(* CoDeSys 2.3.9.59 project: ProgettoSFC.pro *)
(* Libraries: STANDARD.LIB, Iecsfc.lib 12.5.98 13:03:00 *)

(* Task configuration *)
TASK Standard (PRIORITY := 0, INTERVAL := T#10ms);
	MAIN
END_TASK

(* Global variable list: TwinCAT_Configuration *)
(* Generated automatically by TwinCAT - (read only) *)
VAR_CONFIG
	MAIN.tastatore_lettura AT %IB8 : WORD;
END_VAR

(* Data type *)
TYPE ALTEZZA: (nienteA,basso, alto);
END_TYPE

(* Data type *)
TYPE COLORE: (nienteC,rosso, altro);
END_TYPE

(* Data type *)
TYPE PEZZO :
STRUCT
	Colore : COLORE;
	Altezza : ALTEZZA;
	Trapanato:BOOL:=FALSE;
	Tastato:BOOL:=FALSE;
END_STRUCT
END_TYPE

(* Data type *)
TYPE POSTO :
STRUCT
	Presenza :BOOL:=FALSE;
	Pezzo :PEZZO;
END_STRUCT
END_TYPE

(* POU MAIN, SFC *)
PROGRAM MAIN
VAR

(*Variabili Pistone*)
         (*Ingressi*)
	pezzo_magazzino  AT%IX0.0:BOOL; (*sensore che segnala la presenza di un pezzo nel magazzino*)
	pistone_avanti AT%IX0.2:BOOL; (*sensore che segnala se il pistone è avanti*)
	pistone_indietro AT%IX0.4:BOOL; (*sensore che segnala se il pistone è indietro*)
         N_pezzi_spinti: INT:=0; (*variabile che incrementa di 1 quando viene spinto un pezzo sul nastro*)
         (*Uscite*)
	pistone_on  AT%QX0.2:BOOL; (*attuatore del pistone*)



(*Variabili Nastro*)
         (*Ingressi*)
	fine_corsa_nastro  AT%IX0.6:BOOL; (*sensore che segnala il passaggio di un pezzo a fine nastro*)
         (*Uscite*)
	nastro_on  AT%QX0.0:BOOL; (*attuatore del nastro*)


(*Variabili Giostra*)
        Giostra: ARRAY[0..7] OF POSTO;(*array di 8 posti*)
	i: INT :=0; (*indice che incrementa ad ogni movimento della giostra e usato per lavorare con l'array*)
        giostra_busy AT %IX6.1: BOOL; (*sensore che segnala il movimento della giostra*)
        movimento_giostra AT %QX3.4: BOOL; (*attuatore giostra che la muove di 1 posto*)

        T_giostra: TON; (*timer giostra di 2s*)
        mytimegiostra: TIME;
        timer_giostra: BOOL;
        reset_timer_giostra: BOOL;


        T_p1: TON; (*timer buffer 1*)
        mytimep1: TIME;
        timer_p1: BOOL;
        reset_timer_p1: BOOL;

        sensore_colore AT %IX2.1: BOOL; (*sensore che segnala i pezzi di colore rosso*)

        trapano_basso AT %IX2.5: BOOL ; (*sensore che segnala se il trapano è basso*)
        trapano_alto AT %IX2.3: BOOL; (*ensore che segnala se il trapano è alto*)
        trapano_on AT %QX3.7:BOOL; (*attuatore per l'attivazione della punta del trapano*)
        trapano_down AT %QX7.0: BOOL; (*attuatore per fare scendere o salire il trapano*)
        T_trapano: TON; (*timer trapano di 2s*)
        mytimetrapano: TIME;
        timer_trapano: BOOL;
        reset_timer_trapano: BOOL;

        tastatore_basso AT %IX5.3: BOOL; (*sensore che segnala se il tastatore è basso*)
        tastatore_alto AT %IX2.7: BOOL; (*sensore che segnala se il tastatore è alto*)
        tastatore_down AT %QX3.6: BOOL; (*attuatore tastatore*)
	tastatore_lettura AT%I*:WORD; (*fornisce la lettura dell'altezza dei pezzi*)
	(*tastatore_analogico AT %QX4.0: WORD;*)
        T_tastatore: TON; (*timer tastatore di 2s*)
        mytimetastatore: TIME;
        timer_tastatore: BOOL;
        reset_timer_tastatore: BOOL;

        pennarello_alto AT %IX5.4: BOOL; (*sensore che segnala se il pennarello è alto*)
        pennarello_basso AT %IX5.5: BOOL; (*sensore che segnala se il pennarello è basso*)
        pennarello_down AT %QX3.3: BOOL; (*attuatore pennarello*)
        T_pennarello: TON;(*timer pennarello di 2s*)
        mytimepennarello: TIME;
        timer_pennarello: BOOL;
        reset_timer_pennarello: BOOL;

        pistone_PT5_avanti AT %IX5.0: BOOL; (*sensore che segnala se il pistone 5 è avanti*)
        pistone_PT5_indietro AT %IX5.1: BOOL; (*sensore che segnala se il pistone 5 è indietro*)
        pistone_PT5_on AT %QX3.1:BOOL ; (*attuatore pistone 5*)

        pistone_PT6_avanti AT %IX5.7: BOOL;  (*sensore che segnala se il pistone 6 è avanti*)
        pistone_PT6_indietro AT %IX5.6: BOOL; (*sensore che segnala se il pistone 6 è indietro*)
        pistone_PT6_on AT%QX3.5: BOOL; (*attuatore pistone 6*)
        pezzo_baia AT %IX5.2: BOOL; (*sensore che segnala la presenza di un pezzo sulla baia*)


(*Variabili utilizzate nel FOR per la verificare alcune condizioni *)

	j: INT; (*Indice  FOR 1_posto_true*)
	posto_true: BOOL; (*Condizione di ALMENO 1 posto con presenza a TRUE*)

	k: INT; (*Indice  FOR solo_pezzi_rossi*)
	solo_pezzi_rossi: BOOL; (*Condizione SOLO pezzi rossi e  baia occupata*)

	h: INT; (*Indice FOR giostra_piena*)
	giostra_piena: BOOL; (*Condizione TUTTI i pezzi con presenza TRUE*)

	p: INT; (*Indice FOR giostra_vuota*)
	giostra_vuota: BOOL; (*Condizione se ho TUTTI i pezzi con presenza FALSE*) (*forse ridondante*)

	blocco_giostra: BOOL; (*Condizione per bloccare la giostra se ho un pezzo rosso in PT6 e la  baia è già occupata*)

	timer_pistone: BOOL;
	mytimepistone: TIME;
	reset_pistone: BOOL;
	T_pistone: TON;
	T_nastro: TON;
	mytimenastro: TIME;
	timer_nastro: BOOL;
	reset_nastro: BOOL;
	Altezza_tastatore: BOOL;
END_VAR
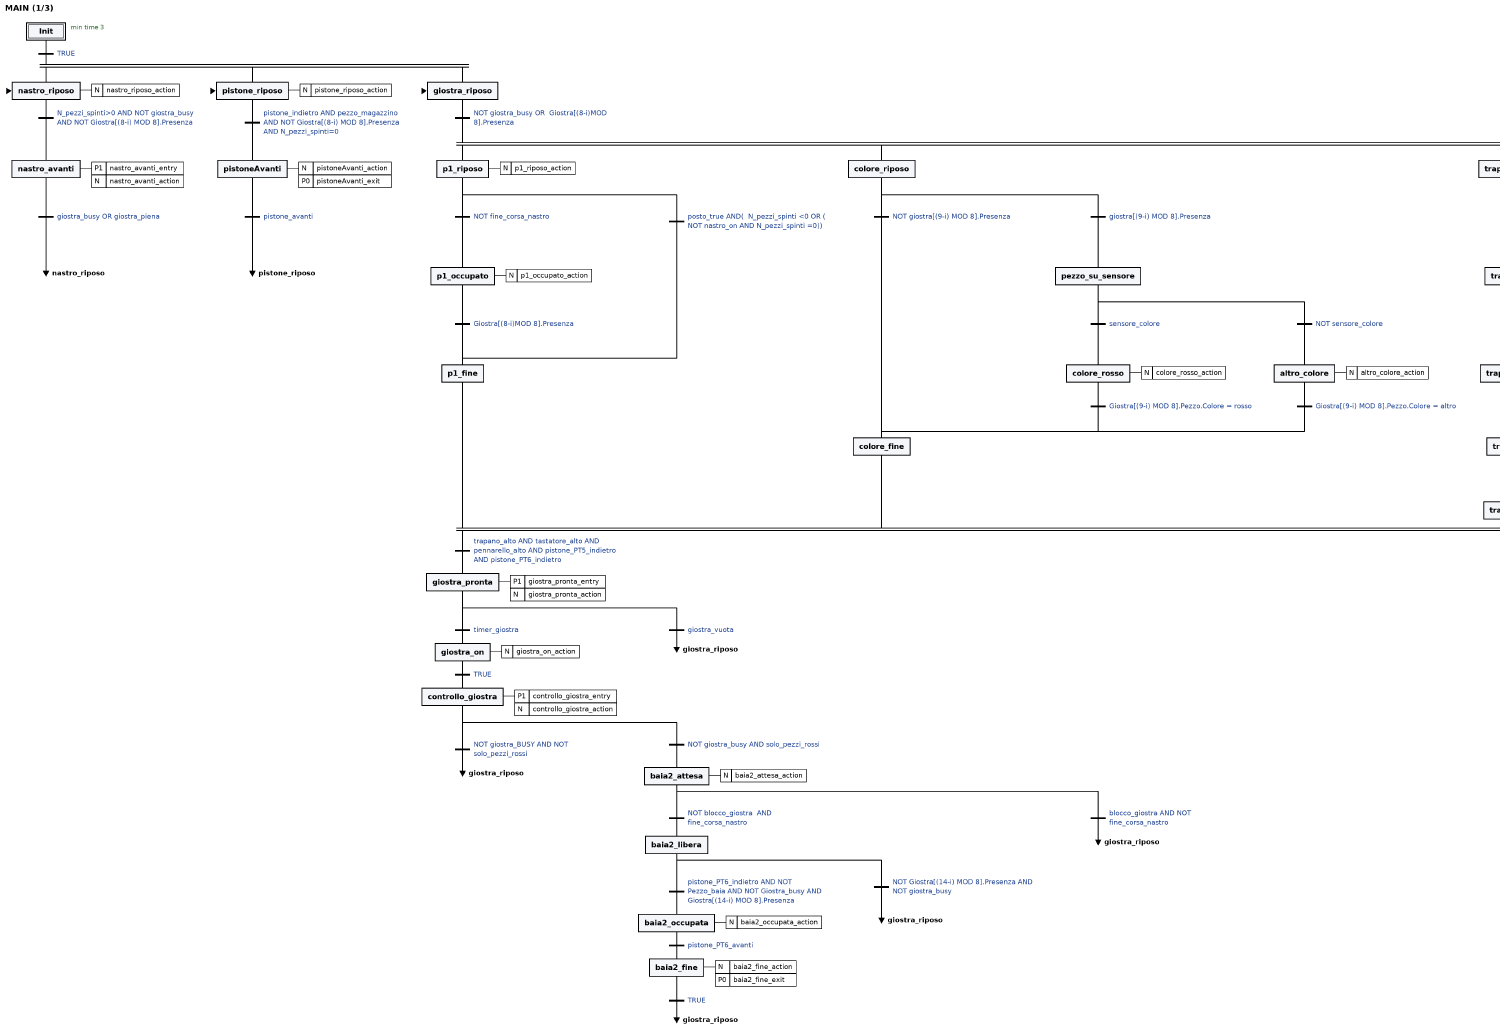
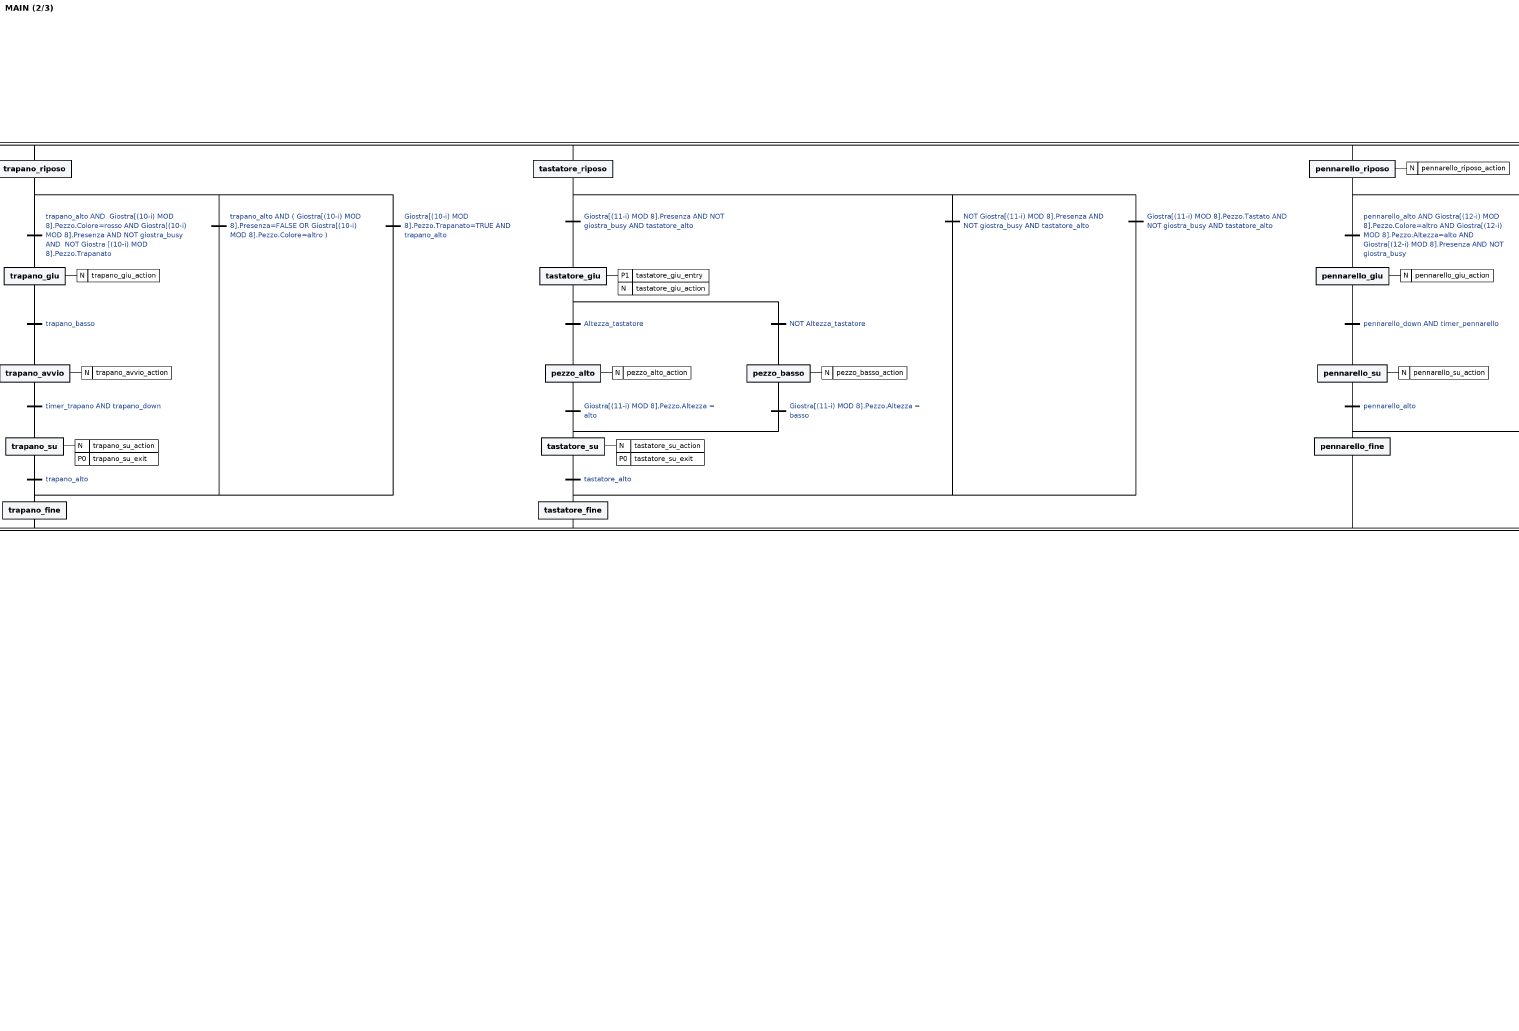
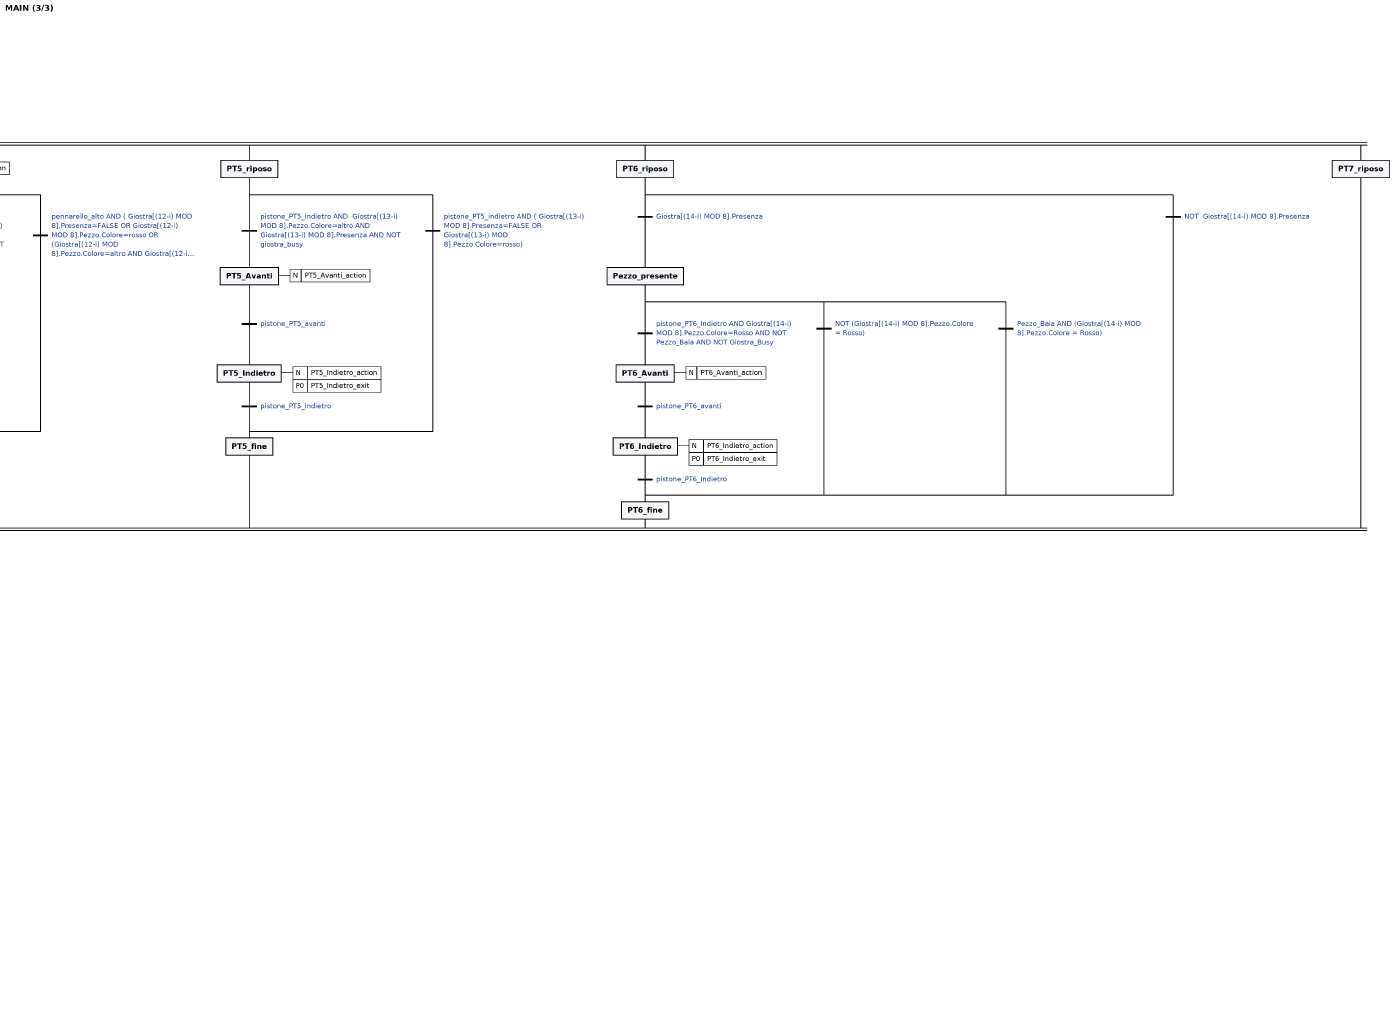
INITIAL_STEP Init: (* min time 3 *)
END_STEP
TRANSITION FROM Init TO (nastro_riposo, pistone_riposo, giostra_riposo) := TRUE;
END_TRANSITION
STEP nastro_riposo:
	nastro_riposo_action(N);
END_STEP
TRANSITION FROM nastro_riposo TO nastro_avanti := N_pezzi_spinti>0 AND NOT giostra_busy AND NOT Giostra[(8-i) MOD 8].Presenza;
END_TRANSITION
STEP pistone_riposo:
	pistone_riposo_action(N);
END_STEP
TRANSITION FROM pistone_riposo TO pistoneAvanti := pistone_indietro AND pezzo_magazzino  AND NOT Giostra[(8-i) MOD 8].Presenza AND N_pezzi_spinti=0;
END_TRANSITION
STEP giostra_riposo:
END_STEP
TRANSITION FROM giostra_riposo TO (p1_riposo, colore_riposo, trapano_riposo, tastatore_riposo, pennarello_riposo, PT5_riposo, PT6_riposo, PT7_riposo) := NOT giostra_busy OR  Giostra[(8-i)MOD 8].Presenza;
END_TRANSITION
STEP p1_riposo:
	p1_riposo_action(N);
END_STEP
TRANSITION FROM p1_riposo TO p1_occupato := NOT fine_corsa_nastro;
END_TRANSITION
TRANSITION FROM p1_riposo TO p1_fine := posto_true AND(  N_pezzi_spinti <0 OR ( NOT nastro_on AND N_pezzi_spinti =0));
END_TRANSITION
STEP p1_occupato:
	p1_occupato_action(N);
END_STEP
TRANSITION FROM p1_occupato TO p1_fine := Giostra[(8-i)MOD 8].Presenza;
END_TRANSITION
STEP p1_fine:
END_STEP
STEP colore_riposo:
END_STEP
TRANSITION FROM colore_riposo TO colore_fine := NOT giostra[(9-i) MOD 8].Presenza;
END_TRANSITION
TRANSITION FROM colore_riposo TO pezzo_su_sensore := giostra[(9-i) MOD 8].Presenza;
END_TRANSITION
STEP pezzo_su_sensore:
END_STEP
TRANSITION FROM pezzo_su_sensore TO colore_rosso := sensore_colore;
END_TRANSITION
TRANSITION FROM pezzo_su_sensore TO altro_colore := NOT sensore_colore;
END_TRANSITION
STEP colore_rosso:
	colore_rosso_action(N);
END_STEP
TRANSITION FROM colore_rosso TO colore_fine := Giostra[(9-i) MOD 8].Pezzo.Colore = rosso;
END_TRANSITION
STEP altro_colore:
	altro_colore_action(N);
END_STEP
TRANSITION FROM altro_colore TO colore_fine := Giostra[(9-i) MOD 8].Pezzo.Colore = altro;
END_TRANSITION
STEP colore_fine:
END_STEP
STEP trapano_riposo:
END_STEP
TRANSITION FROM trapano_riposo TO trapano_giu := trapano_alto AND  Giostra[(10-i) MOD 8].Pezzo.Colore=rosso AND Giostra[(10-i) MOD 8].Presenza AND NOT giostra_busy  AND  NOT Giostra [(10-i) MOD 8].Pezzo.Trapanato;
END_TRANSITION
TRANSITION FROM trapano_riposo TO trapano_fine := trapano_alto AND ( Giostra[(10-i) MOD 8].Presenza=FALSE OR Giostra[(10-i) MOD 8].Pezzo.Colore=altro );
END_TRANSITION
TRANSITION FROM trapano_riposo TO trapano_fine := Giostra[(10-i) MOD 8].Pezzo.Trapanato=TRUE AND trapano_alto;
END_TRANSITION
STEP trapano_giu:
	trapano_giu_action(N);
END_STEP
TRANSITION FROM trapano_giu TO trapano_avvio := trapano_basso;
END_TRANSITION
STEP trapano_avvio:
	trapano_avvio_action(N);
END_STEP
TRANSITION FROM trapano_avvio TO trapano_su := timer_trapano AND trapano_down;
END_TRANSITION
STEP trapano_su:
	trapano_su_action(N);
	trapano_su_exit(P0);
END_STEP
TRANSITION FROM trapano_su TO trapano_fine := trapano_alto;
END_TRANSITION
STEP trapano_fine:
END_STEP
STEP tastatore_riposo:
END_STEP
TRANSITION FROM tastatore_riposo TO tastatore_giu := Giostra[(11-i) MOD 8].Presenza AND NOT giostra_busy AND tastatore_alto;
END_TRANSITION
TRANSITION FROM tastatore_riposo TO tastatore_fine := NOT Giostra[(11-i) MOD 8].Presenza AND NOT giostra_busy AND tastatore_alto;
END_TRANSITION
TRANSITION FROM tastatore_riposo TO tastatore_fine := Giostra[(11-i) MOD 8].Pezzo.Tastato AND NOT giostra_busy AND tastatore_alto;
END_TRANSITION
STEP tastatore_giu:
	tastatore_giu_entry(P1);
	tastatore_giu_action(N);
END_STEP
TRANSITION FROM tastatore_giu TO pezzo_alto := Altezza_tastatore;
END_TRANSITION
TRANSITION FROM tastatore_giu TO pezzo_basso := NOT Altezza_tastatore;
END_TRANSITION
STEP pezzo_alto:
	pezzo_alto_action(N);
END_STEP
TRANSITION FROM pezzo_alto TO tastatore_su := Giostra[(11-i) MOD 8].Pezzo.Altezza = alto;
END_TRANSITION
STEP pezzo_basso:
	pezzo_basso_action(N);
END_STEP
TRANSITION FROM pezzo_basso TO tastatore_su := Giostra[(11-i) MOD 8].Pezzo.Altezza = basso;
END_TRANSITION
STEP tastatore_su:
	tastatore_su_action(N);
	tastatore_su_exit(P0);
END_STEP
TRANSITION FROM tastatore_su TO tastatore_fine := tastatore_alto;
END_TRANSITION
STEP tastatore_fine:
END_STEP
STEP pennarello_riposo:
	pennarello_riposo_action(N);
END_STEP
TRANSITION FROM pennarello_riposo TO pennarello_giu := pennarello_alto AND Giostra[(12-i) MOD 8].Pezzo.Colore=altro AND Giostra[(12-i) MOD 8].Pezzo.Altezza=alto AND Giostra[(12-i) MOD 8].Presenza AND NOT giostra_busy;
END_TRANSITION
TRANSITION FROM pennarello_riposo TO pennarello_fine := pennarello_alto AND ( Giostra[(12-i) MOD 8].Presenza=FALSE OR Giostra[(12-i) MOD 8].Pezzo.Colore=rosso OR (Giostra[(12-i) MOD 8].Pezzo.Colore=altro AND Giostra[(12-i) MOD 8].Pezzo.Altezza=basso));
END_TRANSITION
STEP pennarello_giu:
	pennarello_giu_action(N);
END_STEP
TRANSITION FROM pennarello_giu TO pennarello_su := pennarello_down AND timer_pennarello;
END_TRANSITION
STEP pennarello_su:
	pennarello_su_action(N);
END_STEP
TRANSITION FROM pennarello_su TO pennarello_fine := pennarello_alto;
END_TRANSITION
STEP pennarello_fine:
END_STEP
STEP PT5_riposo:
END_STEP
TRANSITION FROM PT5_riposo TO PT5_Avanti := pistone_PT5_indietro AND  Giostra[(13-i) MOD 8].Pezzo.Colore=altro AND Giostra[(13-i) MOD 8].Presenza AND NOT giostra_busy;
END_TRANSITION
TRANSITION FROM PT5_riposo TO PT5_fine := pistone_PT5_indietro AND ( Giostra[(13-i) MOD 8].Presenza=FALSE OR Giostra[(13-i) MOD 8].Pezzo.Colore=rosso);
END_TRANSITION
STEP PT5_Avanti:
	PT5_Avanti_action(N);
END_STEP
TRANSITION FROM PT5_Avanti TO PT5_Indietro := pistone_PT5_avanti;
END_TRANSITION
STEP PT5_Indietro:
	PT5_Indietro_action(N);
	PT5_Indietro_exit(P0);
END_STEP
TRANSITION FROM PT5_Indietro TO PT5_fine := pistone_PT5_indietro;
END_TRANSITION
STEP PT5_fine:
END_STEP
STEP PT6_riposo:
END_STEP
TRANSITION FROM PT6_riposo TO Pezzo_presente := Giostra[(14-i) MOD 8].Presenza;
END_TRANSITION
TRANSITION FROM PT6_riposo TO PT6_fine := NOT  Giostra[(14-i) MOD 8].Presenza;
END_TRANSITION
STEP Pezzo_presente:
END_STEP
TRANSITION FROM Pezzo_presente TO PT6_Avanti := pistone_PT6_Indietro AND Giostra[(14-i) MOD 8].Pezzo.Colore=Rosso AND NOT Pezzo_Baia AND NOT Giostra_Busy;
END_TRANSITION
TRANSITION FROM Pezzo_presente TO PT6_fine := NOT (Giostra[(14-i) MOD 8].Pezzo.Colore = Rosso);
END_TRANSITION
TRANSITION FROM Pezzo_presente TO PT6_fine := Pezzo_Baia AND (Giostra[(14-i) MOD 8].Pezzo.Colore = Rosso);
END_TRANSITION
STEP PT6_Avanti:
	PT6_Avanti_action(N);
END_STEP
TRANSITION FROM PT6_Avanti TO PT6_Indietro := pistone_PT6_avanti;
END_TRANSITION
STEP PT6_Indietro:
	PT6_Indietro_action(N);
	PT6_Indietro_exit(P0);
END_STEP
TRANSITION FROM PT6_Indietro TO PT6_fine := pistone_PT6_Indietro;
END_TRANSITION
STEP PT6_fine:
END_STEP
STEP PT7_riposo:
END_STEP
TRANSITION FROM (p1_fine, colore_fine, trapano_fine, tastatore_fine, pennarello_fine, PT5_fine, PT6_fine, PT7_riposo) TO giostra_pronta := trapano_alto AND tastatore_alto AND pennarello_alto AND pistone_PT5_indietro AND pistone_PT6_indietro;
END_TRANSITION
STEP giostra_pronta:
	giostra_pronta_entry(P1);
	giostra_pronta_action(N);
END_STEP
TRANSITION FROM giostra_pronta TO giostra_on := timer_giostra;
END_TRANSITION
TRANSITION FROM giostra_pronta TO giostra_riposo := giostra_vuota;
END_TRANSITION
STEP giostra_on:
	giostra_on_action(N);
END_STEP
TRANSITION FROM giostra_on TO controllo_giostra := TRUE;
END_TRANSITION
STEP controllo_giostra:
	controllo_giostra_entry(P1);
	controllo_giostra_action(N);
END_STEP
TRANSITION FROM controllo_giostra TO giostra_riposo := NOT giostra_BUSY AND NOT solo_pezzi_rossi;
END_TRANSITION
TRANSITION FROM controllo_giostra TO baia2_attesa := NOT giostra_busy AND solo_pezzi_rossi;
END_TRANSITION
STEP baia2_attesa:
	baia2_attesa_action(N);
END_STEP
TRANSITION FROM baia2_attesa TO baia2_libera := NOT blocco_giostra  AND fine_corsa_nastro;
END_TRANSITION
TRANSITION FROM baia2_attesa TO giostra_riposo := blocco_giostra AND NOT fine_corsa_nastro;
END_TRANSITION
STEP baia2_libera:
END_STEP
TRANSITION FROM baia2_libera TO baia2_occupata := pistone_PT6_indietro AND NOT Pezzo_baia AND NOT Giostra_busy AND Giostra[(14-i) MOD 8].Presenza;
END_TRANSITION
TRANSITION FROM baia2_libera TO giostra_riposo := NOT Giostra[(14-i) MOD 8].Presenza AND NOT giostra_busy;
END_TRANSITION
STEP baia2_occupata:
	baia2_occupata_action(N);
END_STEP
TRANSITION FROM baia2_occupata TO baia2_fine := pistone_PT6_avanti;
END_TRANSITION
STEP baia2_fine:
	baia2_fine_action(N);
	baia2_fine_exit(P0);
END_STEP
TRANSITION FROM baia2_fine TO giostra_riposo := TRUE;
END_TRANSITION
STEP pistoneAvanti:
	pistoneAvanti_action(N);
	pistoneAvanti_exit(P0);
END_STEP
TRANSITION FROM pistoneAvanti TO pistone_riposo := pistone_avanti;
END_TRANSITION
STEP nastro_avanti:
	nastro_avanti_entry(P1);
	nastro_avanti_action(N);
END_STEP
TRANSITION FROM nastro_avanti TO nastro_riposo := giostra_busy OR giostra_piena;
END_TRANSITION

ACTION nastro_riposo_action:
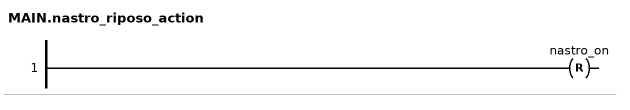
_LD_ (* Ladder Diagram *)
NETWORK 1
	* --- (R nastro_on)
_END_LD_
(* the same logic as Structured Text *)
(* Network 1 *)
nastro_on := FALSE;
END_ACTION

ACTION pistone_riposo_action:
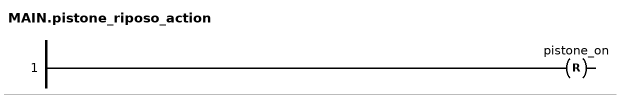
_LD_ (* Ladder Diagram *)
NETWORK 1
	* --- (R pistone_on)
_END_LD_
(* the same logic as Structured Text *)
(* Network 1 *)
pistone_on := FALSE;
END_ACTION

ACTION p1_riposo_action:
FOR j:=0 TO 7 BY 1  DO
IF(Giostra[j].Presenza) THEN posto_true:=TRUE;
EXIT;
ELSE posto_true:=FALSE;
END_IF;


END_FOR;
END_ACTION

ACTION p1_occupato_action:
Giostra[(8-i)MOD 8].Presenza:=TRUE;
N_pezzi_spinti:=N_pezzi_spinti-1;
END_ACTION

ACTION colore_rosso_action:
Giostra[(9-i) MOD 8].Pezzo.Colore := rosso;
END_ACTION

ACTION altro_colore_action:
Giostra[(9-i) MOD 8].Pezzo.Colore := altro;
END_ACTION

ACTION trapano_giu_action:
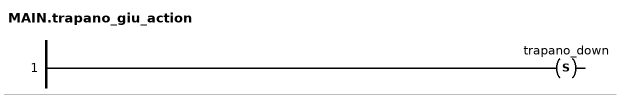
_LD_ (* Ladder Diagram *)
NETWORK 1
	* --- (S trapano_down)
_END_LD_
(* the same logic as Structured Text *)
(* Network 1 *)
trapano_down := TRUE;
END_ACTION

ACTION trapano_avvio_action:
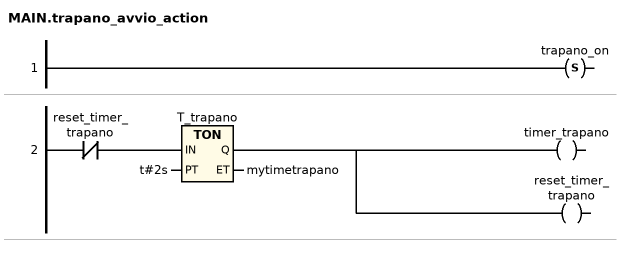
_LD_ (* Ladder Diagram *)
NETWORK 1
	* --- (S trapano_on)
NETWORK 2
	[/reset_timer_trapano] - T_trapano:TON(IN: *, PT: t#2s, ET => mytimetrapano) --- (timer_trapano) (reset_timer_trapano)
_END_LD_
(* the same logic as Structured Text *)
(* Network 1 *)
trapano_on := TRUE;
(* Network 2 *)
T_trapano(IN := NOT reset_timer_trapano, PT := t#2s);
mytimetrapano := T_trapano.ET;
timer_trapano := T_trapano.Q;
reset_timer_trapano := T_trapano.Q;
END_ACTION

ACTION trapano_su_action:
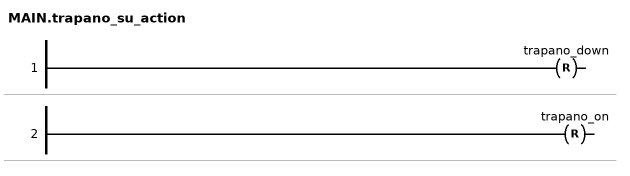
_LD_ (* Ladder Diagram *)
NETWORK 1
	* --- (R trapano_down)
NETWORK 2
	* --- (R trapano_on)
_END_LD_
(* the same logic as Structured Text *)
(* Network 1 *)
trapano_down := FALSE;
(* Network 2 *)
trapano_on := FALSE;
END_ACTION

ACTION trapano_su_exit:
Giostra[(10-i) MOD 8].Pezzo.Trapanato:=TRUE;
END_ACTION

ACTION tastatore_giu_entry:
IF (tastatore_lettura>5)THEN
   Altezza_tastatore := TRUE;
	ELSE
    		Altezza_tastatore := FALSE;
END_IF;
END_ACTION

ACTION tastatore_giu_action:
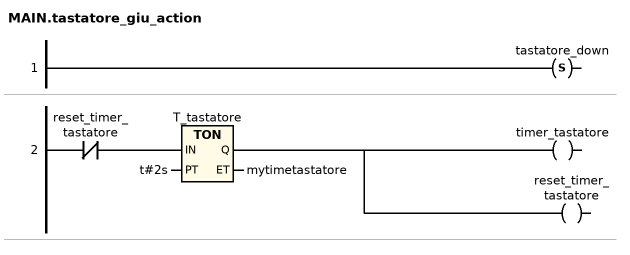
_LD_ (* Ladder Diagram *)
NETWORK 1
	* --- (S tastatore_down)
NETWORK 2
	[/reset_timer_tastatore] - T_tastatore:TON(IN: *, PT: t#2s, ET => mytimetastatore) --- (timer_tastatore) (reset_timer_tastatore)
_END_LD_
(* the same logic as Structured Text *)
(* Network 1 *)
tastatore_down := TRUE;
(* Network 2 *)
T_tastatore(IN := NOT reset_timer_tastatore, PT := t#2s);
mytimetastatore := T_tastatore.ET;
timer_tastatore := T_tastatore.Q;
reset_timer_tastatore := T_tastatore.Q;
END_ACTION

ACTION pezzo_alto_action:
Giostra[(11-i) MOD 8].Pezzo.Altezza:=alto;
END_ACTION

ACTION pezzo_basso_action:
Giostra[(11-i) MOD 8].Pezzo.Altezza:=basso;
END_ACTION

ACTION tastatore_su_action:
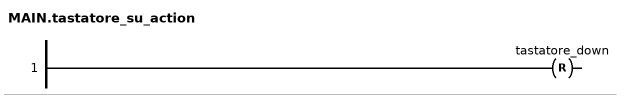
_LD_ (* Ladder Diagram *)
NETWORK 1
	* --- (R tastatore_down)
_END_LD_
(* the same logic as Structured Text *)
(* Network 1 *)
tastatore_down := FALSE;
END_ACTION

ACTION tastatore_su_exit:
Giostra[(11-i) MOD 8].Pezzo.Tastato:=TRUE;
END_ACTION

ACTION pennarello_riposo_action:
IF(Giostra[(12-i) MOD 8].Pezzo.Trapanato) THEN Giostra[(12-i) MOD 8].Pezzo.Colore:=rosso;
END_IF;
END_ACTION

ACTION pennarello_giu_action:
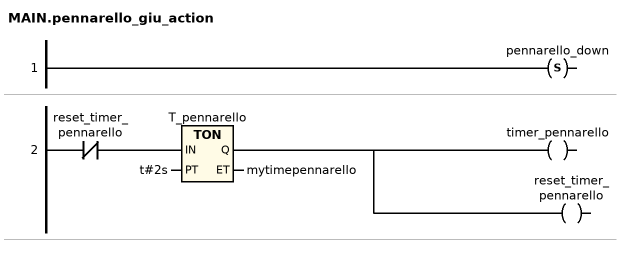
_LD_ (* Ladder Diagram *)
NETWORK 1
	* --- (S pennarello_down)
NETWORK 2
	[/reset_timer_pennarello] - T_pennarello:TON(IN: *, PT: t#2s, ET => mytimepennarello) --- (timer_pennarello) (reset_timer_pennarello)
_END_LD_
(* the same logic as Structured Text *)
(* Network 1 *)
pennarello_down := TRUE;
(* Network 2 *)
T_pennarello(IN := NOT reset_timer_pennarello, PT := t#2s);
mytimepennarello := T_pennarello.ET;
timer_pennarello := T_pennarello.Q;
reset_timer_pennarello := T_pennarello.Q;
END_ACTION

ACTION pennarello_su_action:
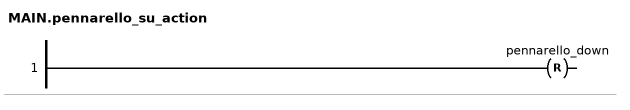
_LD_ (* Ladder Diagram *)
NETWORK 1
	* --- (R pennarello_down)
_END_LD_
(* the same logic as Structured Text *)
(* Network 1 *)
pennarello_down := FALSE;
END_ACTION

ACTION PT5_Avanti_action:
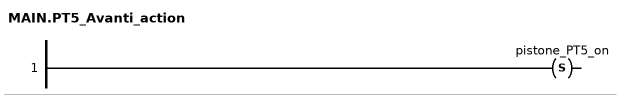
_LD_ (* Ladder Diagram *)
NETWORK 1
	* --- (S pistone_PT5_on)
_END_LD_
(* the same logic as Structured Text *)
(* Network 1 *)
pistone_PT5_on := TRUE;
END_ACTION

ACTION PT5_Indietro_action:
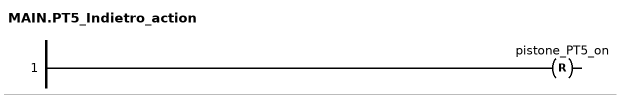
_LD_ (* Ladder Diagram *)
NETWORK 1
	* --- (R pistone_PT5_on)
_END_LD_
(* the same logic as Structured Text *)
(* Network 1 *)
pistone_PT5_on := FALSE;
END_ACTION

ACTION PT5_Indietro_exit:
Giostra[(13-i) MOD 8].Presenza := FALSE;
Giostra[(13-i) MOD 8].Pezzo.Altezza := nienteA;
Giostra[(13-i) MOD 8].Pezzo.Colore := nienteC;
Giostra[(13-i) MOD 8].Pezzo.Tastato := FALSE;
END_ACTION

ACTION PT6_Avanti_action:
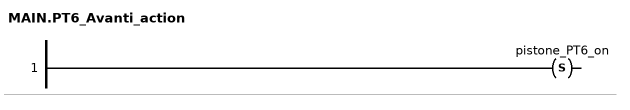
_LD_ (* Ladder Diagram *)
NETWORK 1
	* --- (S pistone_PT6_on)
_END_LD_
(* the same logic as Structured Text *)
(* Network 1 *)
pistone_PT6_on := TRUE;
END_ACTION

ACTION PT6_Indietro_action:
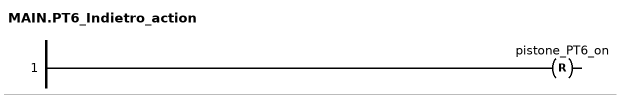
_LD_ (* Ladder Diagram *)
NETWORK 1
	* --- (R pistone_PT6_on)
_END_LD_
(* the same logic as Structured Text *)
(* Network 1 *)
pistone_PT6_on := FALSE;
END_ACTION

ACTION PT6_Indietro_exit:
Giostra[(14-i) MOD 8].Presenza := FALSE;
Giostra[(14-i) MOD 8].Pezzo.Altezza := nienteA;
Giostra[(14-i) MOD 8].Pezzo.Colore := nienteC;
Giostra[(14-i) MOD 8].Pezzo.Trapanato:=FALSE;
Giostra[(14-i) MOD 8].Pezzo.Tastato:=FALSE;
END_ACTION

ACTION giostra_pronta_entry:
(*controlla se il vettore dei posti è vuoto e se è vera attiva la transizione che  rimanda allo stato giostra riposo*)
FOR p:=0 TO 7 BY 1  DO
IF(NOT Giostra[p].Presenza) THEN giostra_vuota:=TRUE;
ELSE giostra_vuota:=FALSE; EXIT;
END_IF;
END_FOR
END_ACTION

ACTION giostra_pronta_action:
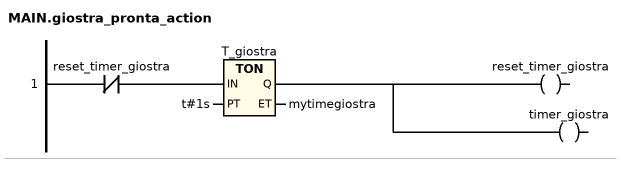
_LD_ (* Ladder Diagram *)
NETWORK 1
	[/reset_timer_giostra] - T_giostra:TON(IN: *, PT: t#1s, ET => mytimegiostra) --- (reset_timer_giostra) (timer_giostra)
_END_LD_
(* the same logic as Structured Text *)
(* Network 1 *)
T_giostra(IN := NOT reset_timer_giostra, PT := t#1s);
mytimegiostra := T_giostra.ET;
reset_timer_giostra := T_giostra.Q;
timer_giostra := T_giostra.Q;
END_ACTION

ACTION giostra_on_action:
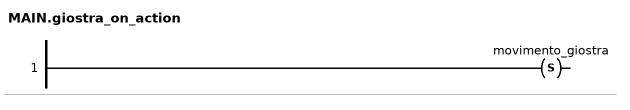
_LD_ (* Ladder Diagram *)
NETWORK 1
	* --- (S movimento_giostra)
_END_LD_
(* the same logic as Structured Text *)
(* Network 1 *)
movimento_giostra := TRUE;
END_ACTION

ACTION controllo_giostra_entry:
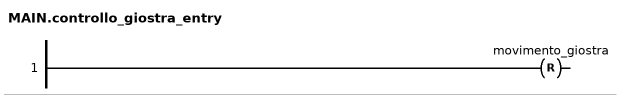
_LD_ (* Ladder Diagram *)
NETWORK 1
	* --- (R movimento_giostra)
_END_LD_
(* the same logic as Structured Text *)
(* Network 1 *)
movimento_giostra := FALSE;
END_ACTION

ACTION controllo_giostra_action:
IF( i=7) THEN i:=0;
ELSE i:=i+1;
END_IF;

(*se la baia è occupata controlla s e ho solo pezzi rossi, se è vera la giostra continua a girare senza utilizzare attuatori (rimanda allo stato giostra_pronta) *)
IF(pezzo_baia=TRUE) THEN

FOR k:=0 TO 7 BY 1  DO
IF(Giostra[k].Pezzo.Colore=rosso  ) THEN solo_pezzi_rossi:=TRUE;
ELSE IF  (Giostra[k].Pezzo.Colore=altro) THEN solo_pezzi_rossi:=FALSE ; EXIT; END_IF;
END_IF;
END_FOR;

END_IF;

(*se la baia non è occupata controlla se ho almeno 1 pezzo NON rosso*)
IF(pezzo_baia=FALSE) THEN

FOR k:=0 TO 7 BY 1  DO
IF(Giostra[k].Pezzo.Colore=altro  ) THEN solo_pezzi_rossi:=FALSE; EXIT; END_IF;
END_FOR;

END_IF
END_ACTION

ACTION baia2_attesa_action:
(*controlla se la baia è occupata e ha davanti un pezzo rosso se è vera blocca tutto*)


IF(pezzo_baia AND Giostra[(14-i) MOD 8].Presenza)
THEN blocco_giostra:=TRUE;

ELSE blocco_giostra:=FALSE;

END_IF;


(*FOR t:=0 TO 7 BY 1  DO
IF(NOT Giostra[t].Pezzo.Trapanato ) THEN lavorati:=FALSE;
ELSE  lavorati:=TRUE ; EXIT;
END_IF;
IF(NOT Giostra[t].Pezzo.Tastato ) THEN lavorati:=FALSE;
ELSE  lavorati:=TRUE ; EXIT;
END_FOR;*)
END_ACTION

ACTION baia2_occupata_action:
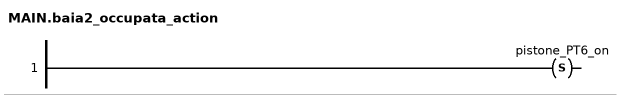
_LD_ (* Ladder Diagram *)
NETWORK 1
	* --- (S pistone_PT6_on)
_END_LD_
(* the same logic as Structured Text *)
(* Network 1 *)
pistone_PT6_on := TRUE;
END_ACTION

ACTION baia2_fine_action:
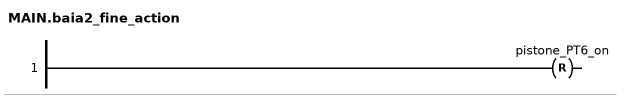
_LD_ (* Ladder Diagram *)
NETWORK 1
	* --- (R pistone_PT6_on)
_END_LD_
(* the same logic as Structured Text *)
(* Network 1 *)
pistone_PT6_on := FALSE;
END_ACTION

ACTION baia2_fine_exit:
Giostra[(14-i) MOD 8].Presenza := FALSE;
Giostra[(14-i) MOD 8].Pezzo.Altezza := nienteA;
Giostra[(14-i) MOD 8].Pezzo.Colore := nienteC;
Giostra[(14-i) MOD 8].Pezzo.Trapanato:=FALSE;
Giostra[(14-i) MOD 8].Pezzo.Tastato:=FALSE;


FOR k:=0 TO 7 BY 1  DO
IF(Giostra[k].Pezzo.Colore=nienteC  ) THEN solo_pezzi_rossi:=FALSE;
ELSE IF (Giostra[k].Pezzo.Colore=rosso  ) THEN solo_pezzi_rossi:=TRUE; EXIT; END_IF;
END_IF
END_FOR;
END_ACTION

ACTION pistoneAvanti_action:
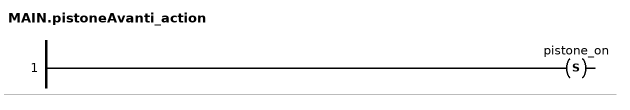
_LD_ (* Ladder Diagram *)
NETWORK 1
	* --- (S pistone_on)
_END_LD_
(* the same logic as Structured Text *)
(* Network 1 *)
pistone_on := TRUE;
END_ACTION

ACTION pistoneAvanti_exit:
N_pezzi_spinti:=N_pezzi_spinti+1;
END_ACTION

ACTION nastro_avanti_entry:
FOR h:=0 TO 7 BY 1  DO
IF(Giostra[h].Presenza) THEN giostra_piena:=TRUE;
ELSE giostra_piena:=FALSE; EXIT;
END_IF;

END_FOR;
END_ACTION

ACTION nastro_avanti_action:
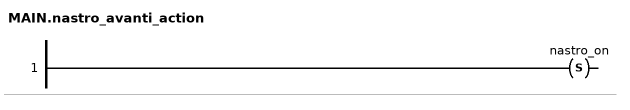
_LD_ (* Ladder Diagram *)
NETWORK 1
	* --- (S nastro_on)
_END_LD_
(* the same logic as Structured Text *)
(* Network 1 *)
nastro_on := TRUE;
END_ACTION
END_PROGRAM
